{attribute 'GeneratedUsingTerminal: EL9505-0000-0016'}
{attribute addProperty BoxType "EL9505-0000-0016"}
{attribute addProperty Id "Power_OKAT %I*BOOL1OverloadAT %I*BOOL1"}
{attribute addProperty CRC "3101291258"}
{attribute addProperty Size "2"}
TYPE Status_Uo_B8D9F2FA :
STRUCT
	{attribute addProperty Name "Power_OK"}
	Power_OK AT %I* : BOOL;
	{attribute addProperty Name "Overload"}
	Overload AT %I* : BOOL;
END_STRUCT
END_TYPE

(* stored: Version 1.2.0.0, ProductVersion 3.1.4024.9
   DUT Status_Uo_B8D9F2FA: Id {bc8cc477-740d-443e-aaa9-2f1ed3044579} *)
